Staubli VAL3: OnF6.pgx

program OnF6()
  local string l_sTemp
begin
  //参数
  call setPara()
end
